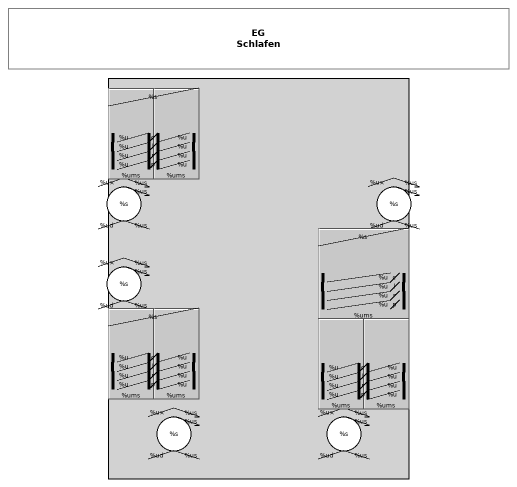
[picture p24: VI_SCHLAFEN (HMI screen)]
rectangle at (130,0)-(631,61): text "EG / Schlafen"
embedded screen at (440,400)-(491,451): vi_Lamp
embedded screen at (490,170)-(541,221): vi_Lamp
embedded screen at (270,400)-(321,451): vi_Lamp
embedded screen at (220,250)-(271,301): vi_Lamp
embedded screen at (220,170)-(271,221): vi_Lamp
embedded screen at (440,220)-(531,401): vi_ButtonTripple
embedded screen at (230,300)-(321,391): vi_ButtonDouble
embedded screen at (230,80)-(321,171): vi_ButtonDouble
1 more shapes without text or variables
*)

(* Visualisation templates/vi_Smoke
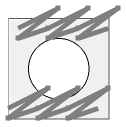
button at (0,0)-(101,101): taps $fbMotiondetector$.viIN
ellipse at (20,20)-(81,81): alarm colour if $fbMotiondetector$.myIN; taps $fbMotiondetector$.viIN
2 more shapes without text or variables
*)

(* Visualisation EG/VI_SPEIS
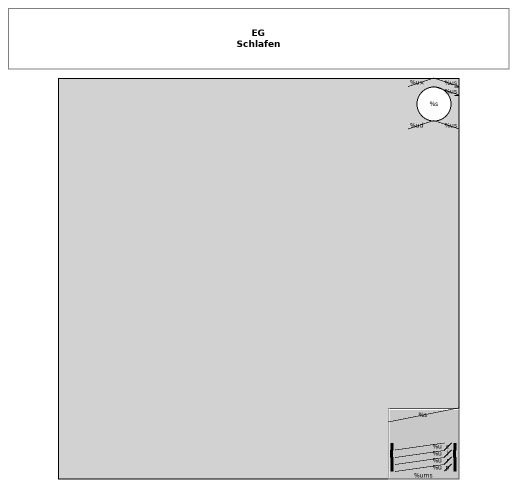
rectangle at (130,0)-(631,61): text "EG / Schlafen"
embedded screen at (530,70)-(581,121): vi_Lamp
embedded screen at (510,400)-(581,471): vi_ButtonSingle
1 more shapes without text or variables
*)

(* Visualisation templates/VI_TEMPERATURE
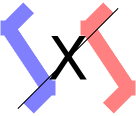
polyline at (0,0)-(100,100): text "X"; invisible if NOT $fb_Temperature$.Error
2 more shapes without text or variables
1 elements of other kinds (tables, trends, ...) not read
*)

(* Visualisation VI_Temperaturen
rectangle at (130,0)-(631,61): text "Temperaturen"
1 elements of other kinds (tables, trends, ...) not read
*)

(* Visualisation KG/VI_VORRAT
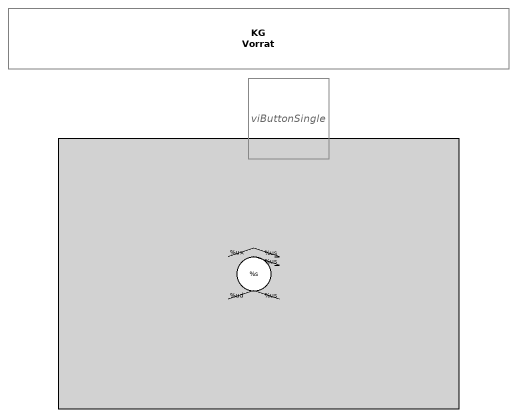
rectangle at (130,0)-(631,61): text "KG / Vorrat"
embedded screen at (350,240)-(401,291): vi_Lamp
embedded screen at (370,70)-(451,151): viButtonSingle
1 more shapes without text or variables
*)

(* Visualisation KG/VI_WASCHEN
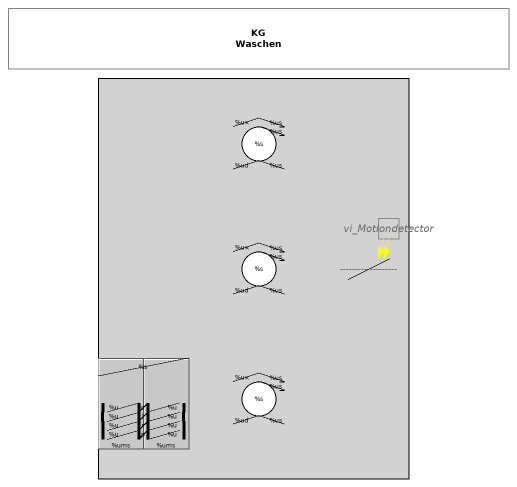
rectangle at (130,0)-(631,61): text "KG / Waschen"
embedded screen at (220,350)-(311,441): vi_ButtonDouble
embedded screen at (355,235)-(406,286): vi_Lamp
embedded screen at (355,365)-(406,416): vi_Lamp
embedded screen at (355,110)-(406,161): vi_Lamp
embedded screen at (500,210)-(521,231): vi_Motiondetector
embedded screen at (470,230)-(511,271): vi_Light
1 more shapes without text or variables
*)
